FUNCTION_BLOCK HistorianFunctionBlock
VAR_INPUT
	
END_VAR

VAR_OUTPUT
	
END_VAR

VAR
	HistorianStateMachine			:	UINT	:=	3;
	
	FIFO_Buffer_In_Modbus			:	ARRAY [0..1199] OF EventRecorder_In_Modbus;
	FIFO_Buffer_In_EAP 				:	ARRAY [0..1199] OF EventRecorder_In_EAP;
	FIFO_Buffer_ControllerOut 		:	ARRAY [0..1199] OF EventRecorder_Controller_Output;
	FIFO_Buffer_Index_TimeStamp		:	ARRAY [0..1199] OF Index_TimeStamp;	
	
	
	FIFO_Transmit_EAP_Index			:	INT;
	FIFO_Transmit_Modbus_Index		:	INT;
	FIFO_Transmit_ControlOut_Index	:	INT;
	
	
	FIFO_Index_Max					:	INT := 1200;
	PreEventCaptures				:	INT	:= 200;	// 20 Percent of preevent recored
	
	FIFO_StopIndex					:	INT;
	FIFO_StopIndex_Modbus			:	INT;
	FIFO_StopIndex_ControlOut		:	INT;
	
	FIFO_index						:	INT;
	FIFO_index_Modbus				:	INT;
	FIFO_index_ControlOut			:	INT;
	
	
	TranmitingIndex					:	INT;
	RecordingTriger					:	BOOL;
	_TransmitRequest				:	INT;
	FIFO_Transmit_Index				:	INT;
	
	EAP_Record_done			:	BOOL := FALSE;
	Modbus_Record_done		:	BOOL := FALSE;
	ControlOut_Record_done	:	BOOL := FALSE;
	
	EAP_trigger_done		:	BOOL := FALSE;
	Modbus_triger_done		:	BOOL := FALSE;
	ControlOut_triger_done	:	BOOL := FALSE;
		
	unixTime: UnixTimestamp;
    timestampSeconds: ULINT;
    timestampMilliseconds: ULINT;
	

END_VAR

PROPERTY GetRequest : INT;
GET
GetRequest	:=	_TransmitRequest;
END_GET
END_PROPERTY

METHOD PUBLIC ListeningRecording_ControlOut : BOOL
VAR_INPUT
	HistorianDataPacket		:	EventRecorder_Controller_Output;
END_VAR

VAR_OUTPUT
	
END_VAR

VAR
	icounter	:	INT;
END_VAR
// State machine for Historian
IF EAP_trigger_done AND NOT ControlOut_triger_done AND RecordingTriger THEN
	// Set stop index with buffer wrapping
		FIFO_StopIndex_ControlOut := FIFO_index_ControlOut - PreEventCaptures;	//	Set the end of FIFO buffer
		IF FIFO_StopIndex_ControlOut < 0 THEN							// wrapping
			FIFO_StopIndex_ControlOut := FIFO_Index_Max + FIFO_StopIndex_ControlOut;
		END_IF
		// Go to the recording State
		HistorianStateMachine := 1;
		ControlOut_triger_done := TRUE;
END_IF
CASE HistorianStateMachine	OF
//---------------- Begin of Listening State -------------------------------	
	0:	// Listening
		FIFO_index_ControlOut := FIFO_index_ControlOut + 1;							// Inceasing buffer index
		IF FIFO_index_ControlOut = FIFO_Index_Max THEN						// Buffer wrapping
			FIFO_index_ControlOut := 0;
		END_IF	
	
		FIFO_Buffer_ControllerOut[FIFO_index_ControlOut] := HistorianDataPacket;			// Copy data to buffer
		
		IF RecordingTriger = TRUE AND NOT ControlOut_triger_done THEN
			// Set stop index with buffer wrapping
			FIFO_StopIndex_ControlOut := FIFO_index_ControlOut - PreEventCaptures;	//	Set the end of FIFO buffer
			IF FIFO_StopIndex_ControlOut < 0 THEN							// wrapping
				FIFO_StopIndex_ControlOut := FIFO_Index_Max + FIFO_StopIndex_ControlOut;
			END_IF
			// Go to the recording State
			HistorianStateMachine := 1;
		END_IF
//---------------- End of Listening State   -------------------------------	

//---------------- Begin of Recording State -------------------------------		
	1:	
		IF NOT ControlOut_Record_done THEN
	
			FIFO_index_ControlOut := FIFO_index_ControlOut + 1;					// Inceasing buffer index
			IF FIFO_index_ControlOut = FIFO_Index_Max THEN				// Buffer wrapping
				FIFO_index_ControlOut := 0;
			END_IF
			
			FIFO_Buffer_ControllerOut[FIFO_index_ControlOut] := HistorianDataPacket;	
			
			IF FIFO_index_ControlOut = FIFO_StopIndex_ControlOut THEN				// change to transmit state
				ControlOut_Record_done	:= TRUE;					// Send request
			END_IF
		END_IF
		
	3: // Initialization
		FOR icounter :=	0 TO (FIFO_Index_Max-1)	BY 1 DO
			FIFO_Buffer_Index_Timestamp[icounter].Index := icounter;
		END_FOR
		HistorianStateMachine := 0;
END_CASE
END_METHOD

METHOD PUBLIC ListeningRecording_IN_EAP : BOOL
VAR_INPUT
	HistorianDataPacket		:	EventRecorder_In_EAP;
END_VAR

VAR_OUTPUT
	
END_VAR

VAR
	icounter	:	INT;
END_VAR
// State machine for Historian

CASE HistorianStateMachine	OF
//---------------- Begin of Listening State -------------------------------	
	0:	// Listening
		FIFO_index := FIFO_index + 1;							// Inceasing buffer index
		IF FIFO_index = FIFO_Index_Max THEN						// Buffer wrapping
			FIFO_index := 0;
		END_IF	
	
		FIFO_Buffer_In_EAP[FIFO_index] := HistorianDataPacket;			// Copy data to buffer
		
		IF RecordingTriger = TRUE AND NOT EAP_trigger_done THEN
			// Set stop index with buffer wrapping
			FIFO_StopIndex := FIFO_index - PreEventCaptures;	//	Set the end of FIFO buffer
			IF FIFO_StopIndex < 0 THEN							// wrapping
				FIFO_StopIndex := FIFO_Index_Max + FIFO_StopIndex;
			END_IF
			// Go to the recording State
			EAP_trigger_done := TRUE;
			HistorianStateMachine := 1;
		END_IF
//---------------- End of Listening State   -------------------------------	

//---------------- Begin of Recording State -------------------------------		
	1:	
		
		IF NOT EAP_Record_done THEN
	
			FIFO_index := FIFO_index + 1;					// Inceasing buffer index
			IF FIFO_index = FIFO_Index_Max THEN				// Buffer wrapping
				FIFO_index := 0;
			END_IF
			
			FIFO_Buffer_In_EAP[FIFO_index] := HistorianDataPacket;	
			
			IF FIFO_index = FIFO_StopIndex THEN				// change to transmit state
				EAP_Record_done	:= TRUE;					// Send request
			END_IF
		END_IF
		
	3: // Initialization
		FOR icounter :=	0 TO (FIFO_Index_Max-1)	BY 1 DO
			FIFO_Buffer_Index_Timestamp[icounter].Index := icounter;
		END_FOR
		HistorianStateMachine := 0;
END_CASE
END_METHOD

METHOD ListeningRecording_IN_Modbus : BOOL
VAR_INPUT
	HistorianDataPacket		:	EventRecorder_In_Modbus;
END_VAR

VAR_OUTPUT
	
END_VAR

VAR
	icounter	:	INT;
END_VAR
// Unix Time
Globalvar.unixTime();
Globalvar.timestampMilliseconds := ULINT_TO_UINT(Globalvar.unixTime.milliseconds - Globalvar.unixTime.seconds*1000);
Globalvar.timestampSeconds.dwSecond := ULINT_TO_DWORD(Globalvar.unixTime.seconds);


// State machine for Historian
IF EAP_trigger_done AND NOT Modbus_Triger_done AND RecordingTriger THEN
	// Set stop index with buffer wrapping
			FIFO_StopIndex_Modbus := FIFO_index_Modbus - PreEventCaptures;	//	Set the end of FIFO buffer
			IF FIFO_StopIndex_Modbus < 0 THEN								// wrapping
				FIFO_StopIndex_Modbus := FIFO_Index_Max + FIFO_StopIndex_Modbus;
			END_IF
			// Go to the recording State
			HistorianStateMachine := 1;
			Modbus_Triger_done := TRUE;
END_IF
CASE HistorianStateMachine	OF
//---------------- Begin of Listening State -------------------------------	
	0:	// Listening
		FIFO_index_Modbus := FIFO_index_Modbus + 1;							// Inceasing buffer index
		IF FIFO_index_Modbus = FIFO_Index_Max THEN						// Buffer wrapping
			FIFO_index_Modbus := 0;
		END_IF	
	
		FIFO_Buffer_In_Modbus[FIFO_index_Modbus] := HistorianDataPacket;			// Copy data to buffer
		FIFO_Buffer_Index_TimeStamp[FIFO_index_Modbus].TimeStamp := Globalvar.timestampSeconds.dtSecond;
		FIFO_Buffer_Index_TimeStamp[FIFO_index_Modbus].Miliseconds := Globalvar.timestampMilliseconds;
		
		IF RecordingTriger = TRUE AND NOT Modbus_triger_done  THEN
			// Set stop index with buffer wrapping
			FIFO_StopIndex_Modbus := FIFO_index_Modbus - PreEventCaptures;	//	Set the end of FIFO buffer
			IF FIFO_StopIndex_Modbus < 0 THEN								// wrapping
				FIFO_StopIndex_Modbus := FIFO_Index_Max + FIFO_StopIndex_Modbus;
			END_IF
			// Go to the recording State
			HistorianStateMachine := 1;
		END_IF
//---------------- End of Listening State   -------------------------------	

//---------------- Begin of Recording State -------------------------------		
	1:	IF NOT 	Modbus_Record_done THEN
		
			FIFO_index_Modbus := FIFO_index_Modbus + 1;					// Inceasing buffer index
			IF FIFO_index_Modbus = FIFO_Index_Max THEN				// Buffer wrapping
				FIFO_index_Modbus := 0;
			END_IF
			
			FIFO_Buffer_In_Modbus[FIFO_index_Modbus] := HistorianDataPacket;	
			FIFO_Buffer_Index_TimeStamp[FIFO_index_Modbus].TimeStamp := Globalvar.timestampSeconds.dtSecond;
			FIFO_Buffer_Index_TimeStamp[FIFO_index_Modbus].Miliseconds := Globalvar.timestampMilliseconds;
			
			IF FIFO_index_Modbus = FIFO_StopIndex_Modbus THEN	// change to transmit state
				Modbus_Record_done := TRUE;						// Send request
			END_IF
		END_IF
END_CASE
END_METHOD

PROPERTY SetTtriger : BOOL
SET
RecordingTriger := SetTtriger;
END_SET
END_PROPERTY

METHOD PUBLIC Transmiting : BOOL
VAR_INPUT
	
END_VAR

VAR_OUTPUT
	HistorianDataPacket_EtherCAT	:	EthercatDataPacket;
END_VAR
IF EAP_Record_done AND Modbus_Record_done  AND ControlOut_Record_done THEN
	_TransmitRequest := 1;
	HistorianStateMachine := 2;
ELSE
	_TransmitRequest := 0;
END_IF

// State machine for Historian
CASE HistorianStateMachine	OF
//---------------- Begin of Transmiting State -----------------------------	
	2:
		IF gvl.TransmitApproved = 1  THEN
			
		// Increasing transmitting index
			FIFO_Transmit_Index := FIFO_Transmit_Index + 1;
		
			FIFO_Transmit_EAP_Index := FIFO_index + FIFO_Transmit_Index;
			FIFO_Transmit_Modbus_Index := FIFO_index_Modbus + FIFO_Transmit_Index;
			FIFO_Transmit_ControlOut_Index := FIFO_index_ControlOut + FIFO_Transmit_Index;
			
			IF FIFO_Transmit_EAP_Index >= FIFO_Index_Max THEN					// Buffer wrapping
				FIFO_Transmit_EAP_Index := FIFO_Transmit_EAP_Index - FIFO_Index_Max;
			END_IF
			
			IF FIFO_Transmit_Modbus_Index >= FIFO_Index_Max THEN					// Buffer wrapping
				FIFO_Transmit_Modbus_Index := FIFO_Transmit_Modbus_Index - FIFO_Index_Max;
			END_IF
			
			IF FIFO_Transmit_ControlOut_Index >= FIFO_Index_Max THEN					// Buffer wrapping
				FIFO_Transmit_ControlOut_Index := FIFO_Transmit_ControlOut_Index - FIFO_Index_Max;
			END_IF
			
			HistorianDataPacket_EtherCAT.SingalIn_Modbus := FIFO_Buffer_In_Modbus[FIFO_Transmit_Modbus_Index];		// Map to EtherCAT
			HistorianDataPacket_EtherCAT.SignalIn_EAP := FIFO_Buffer_In_EAP[FIFO_Transmit_EAP_Index];			// Map to EtherCAT
			HistorianDataPacket_EtherCAT.ControllerOut := FIFO_Buffer_ControllerOut[FIFO_Transmit_ControlOut_Index];
			HistorianDataPacket_EtherCAT.Index_TimeStamp.Index := FIFO_Transmit_Index - 1;
			
			HistorianDataPacket_EtherCAT.Index_TimeStamp.TimeStamp := FIFO_Buffer_Index_TimeStamp[FIFO_Transmit_Modbus_Index].TimeStamp ;
			HistorianDataPacket_EtherCAT.Index_TimeStamp.Miliseconds := FIFO_Buffer_Index_TimeStamp[FIFO_Transmit_Modbus_Index].Miliseconds;
			
			// Done and Switch to listening State
			IF FIFO_Transmit_Index >= FIFO_Index_Max THEN
				FIFO_Transmit_Index := 0;		// Remove request
				HistorianStateMachine := 0;
				
				FIFO_index := 0;
				FIFO_index_Modbus := 0;
				FIFO_index_ControlOut := 0;
				
				EAP_Record_done := FALSE;
				Modbus_Record_done	:=	FALSE;
				ControlOut_Record_done := FALSE;
				
				EAP_trigger_done := FALSE;
				Modbus_Triger_done := FALSE;
				ControlOut_triger_done := FALSE;
				
			END_IF			
		END_IF
//---------------- End of Transmiting State -------------------------------	
END_CASE
END_METHOD

END_FUNCTION_BLOCK

(* stored: Version 1.1.0.1
   POU HistorianFunctionBlock: Id {e47bf73b-626d-49fa-8f07-412b7ee0fdf6}, SpecialFunc None
   Property GetRequest: Id {658e5794-fd97-4169-a6b3-d5c247dc9f6e}
   Get Get: Id {cee7bc8c-cdc0-4f3c-9857-15490bcf58d6}
   Method ListeningRecording_ControlOut: Id {deba191c-c01d-4985-b7eb-6d5d49360102}
   Method ListeningRecording_IN_EAP: Id {527bd702-ad0c-437b-bc86-b07c54b925a8}
   Method ListeningRecording_IN_Modbus: Id {84023060-3153-49b5-942c-da97b10a7bbe}
   Property SetTtriger: Id {7787d145-e19d-43cf-afe8-0d79864c4861}
   Set Set: Id {f4b42821-2592-4b8d-a46f-b45f8486b56f}
   Method Transmiting: Id {e7f7d31f-63bc-4223-8795-541f0c9fd1a9} *)
